{attribute 'GeneratedUsingTerminal: EK1100-0000-0018'}
{attribute addProperty BoxType "EK1100-0000-0018"}
{attribute addProperty Id "Beckhoff_BKxxxxEK1122Beckhoff_BKxxxxEK1122_C32C6A5C0A_0015_BK1250_0000_0016A_0015_BK1250_0000_0016_5F4E76F70"}
{attribute addProperty CRC "1934701483"}
{attribute addProperty Size "0"}
TYPE Beckhoff_BKxxxx_735133AB EXTENDS EK1100_1FC0878B :
STRUCT
	{attribute addProperty Name "Beckhoff_BKxxxxEK1122"}
	{attribute addProperty PreviousPort "Beckhoff BKxxxx : B"}
	Beckhoff_BKxxxxEK1122 : Beckhoff_BKxxxxEK1122_C32C6A5C;
	{attribute addProperty Name "A_0015_BK1250_0000_0016"}
	{attribute addProperty PreviousPort "Beckhoff BKxxxxEK1122 : C"}
	A_0015_BK1250_0000_0016 : A_0015_BK1250_0000_0016_5F4E76F7;
END_STRUCT
END_TYPE

(* stored: Version 1.2.0.0, ProductVersion 3.1.4024.9
   DUT Beckhoff_BKxxxx_735133AB: Id {96cc7e59-e62b-404c-9cf6-693e4f69c27b} *)
